{attribute 'qualified_only'}
{attribute 'analysis' := '-33'}
VAR_GLOBAL
	{attribute 'OPC.UA.DA' := '1'}
	MonitorTestData		: MonitorTest;
	{attribute 'OPC.UA.DA' := '1'}
	ReadTestData		: ReadTest;
	{attribute 'OPC.UA.DA' := '1'}
	SymbolTestData		: SymbolTest;
	{attribute 'OPC.UA.DA' := '1'}
	WriteTestData		: WriteTest;
END_VAR

(* stored: Version 1.1.0.1
   GVL OpcNet9: Id {65acbbf4-22b6-0840-1b27-53986e46b206} *)
